// Mitsubishi GX Works2 project: PLC 카운터 (자동 리셋1)   PLC: Q03UDV

PROGRAM MAIN
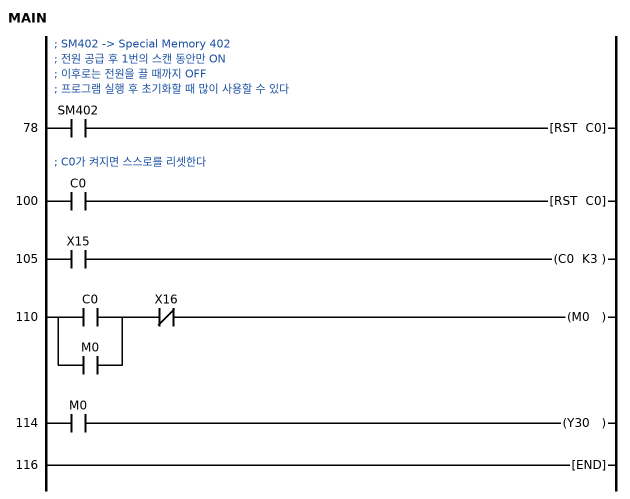
; SM402 -> Special Memory 402
; 전원 공급 후 1번의 스캔 동안만 ON
; 이후로는 전원을 끌 때까지 OFF
; 프로그램 실행 후 초기화할 때 많이 사용할 수 있다
78    LD      SM402
      RST     C0
; C0가 켜지면 스스로를 리셋한다
100   LD      C0
      RST     C0
105   LD      X15
      OUT     C0 K3
110   LD      C0
      OR      M0
      ANI     X16
      OUT     M0
114   LD      M0
      OUT     Y30
116   END
END_PROGRAM
